{attribute 'qualified_only'}
{attribute 'strict'}
{attribute 'to_string'}
TYPE PieceType_e :
(
	long,
	short,
	_max
);
END_TYPE

(* stored: Version 1.1.0.1, ProductVersion 3.1.4024.6
   EnumerationTextList PieceType_e: Id {4c0546ef-5046-429b-b703-8ba5048646cb} *)
